FUNCTION F_BlockCopy : BOOL
VAR_INPUT
	pSrc	: PVOID;
	LenSrc  : UDINT;
	pDest 	: PVOID;
	LenDest	: UDINT;
END_VAR

VAR

END_VAR


IF LenSrc > 0 AND
   LenDest > 0 AND
   pSrc > 0 AND
   pDest > 0 THEN 
	
	MEMSET(destAddr := pDest, 0, LenDest);
   
	IF LenSrc > LenDest THEN	
		MEMCPY(destAddr := pDest, srcAddr := pSrc, n := LenDest);
	ELSE
		MEMCPY(destAddr := pDest, srcAddr := pSrc, n := LenSrc);
	END_IF

	F_BlockCopy := TRUE;
ELSE
	F_BlockCopy := FALSE;
END_IF

END_FUNCTION

(* stored: Version 1.1.0.1, ProductVersion 3.1.4020.6
   POU F_BlockCopy: Id {931f677d-4574-4f16-b58f-81218aff8ae8}, SpecialFunc None *)
